# EPICS substitutions: modules/event/evrSupport/Db/ioc/IOC-LI25-PM01evr.substitutions
#==============================================================================
#
# Abs:  LCLS EVR IOC records for LI25 PM01
#
# Name: IOC-LI25-PM01evr.substitutions
#
#==============================================================================
#
file evrPMXX.db
{
pattern { DEVICE        }
	{ EVR:LI25:PM01 }
}
